{attribute 'qualified_only'}
{attribute 'strict'}
TYPE eColors :
(
	red := 16#FFFF0000,
	green := 16#FF00FF00,
	blue := 16#FF0000FF,
	orange := 16#FFFF8000
)DWORD;
END_TYPE

(* stored: Version 1.1.0.1, ProductVersion 3.1.4024.11
   DUT eColors: Id {f10dbe01-0865-4046-9916-0790b41872ee} *)
